FUNCTION_BLOCK ServoAxis EXTENDS ParentAxis
VAR
	
	_AxisReference				: AXIS_REF;
	
	_Enable						: MC_Power;
	_ReadStatus					: MC_ReadStatus;
	_Reset						: MC_Reset;
	_MoveRelative				: MC_MoveRelative;
	
	_Status						: NcAxisRefStatus;
	
END_VAR

METHOD CyclicUpdate : HRESULT
VAR_INPUT
END_VAR

_ClassRunningIndicatorToggle := NOT(_ClassRunningIndicatorToggle);

_Enable(Axis := _AxisReference);
_Reset(Axis := _AxisReference);
_MoveRelative(Axis := _AxisReference);

_ReadStatus
(
	Axis 					:= _AxisReference,
	Enable 					:= TRUE,
	Error 					=> _Status._Error,
	ErrorID 				=> _Status._ErrorID,
	ErrorStop 				=> _Status._ErrorStop,
	Disabled 				=> _Status._Disabled,
	Stopping 				=> _Status._Stopping,
	StandStill 				=> _Status._StandStill,
	DiscreteMotion 			=> _Status._DiscreteMotion,
	ContinuousMotion 		=> _Status._ContinuousMotion,
	SynchronizedMotion 		=> _Status._SynchronizedMotion,
	Homing 					=> _Status._Homing,
	ConstantVelocity 		=> _Status._ConstantVelocity,
	Accelerating 			=> _Status._Accelerating,
	Decelerating 			=> _Status._Decelerating,
	Status 					=> _Status._Status
);

_IsBusyMoving :=
(
	_ReadStatus.DiscreteMotion OR
	_ReadStatus.ConstantVelocity OR
	_ReadStatus.SynchronizedMotion
);

_IsBusyStopping :=
(
	_ReadStatus.Stopping
);

_IsReadyForCommand :=
(
	NOT(_ReadStatus.Disabled) AND
	NOT(_IsBusyMoving) AND
	NOT(_IsBusyStopping) AND
	NOT(_ReadStatus.Error) AND
	NOT(_ReadStatus.ErrorStop)
);

_IsDoneWithCommand :=
(
	_Reset.Done OR
	_MoveRelative.Done
);

_IsInError :=
(
	_ReadStatus.Error
);

_CurrentErrorCode := _ReadStatus.ErrorID;
	
IF _Status._ErrorID <> 0 THEN
	_PreviousErrorCode := _ReadStatus.ErrorID;
END_IF

_ErrorRTrig(CLK := _IsInError);
IF _ErrorRTrig.Q THEN
	_ErrorCount := _ErrorCount + 1;
END_IF


CyclicUpdate := 1;
RETURN;
END_METHOD

METHOD StartDisable : BOOL
_Enable(Axis := _AxisReference);

_Enable.Enable := FALSE;
_Enable.Enable_Negative := FALSE;
_Enable.Enable_Positive := FALSE;
_Enable.Override := 0;

IF NOT(_Enable.Status) THEN
	StartDisable := TRUE;
	RETURN;
ELSE
	;
END_IF

RETURN;
END_METHOD

METHOD StartEnable : BOOL
_Enable(Axis := _AxisReference);

_Enable.Enable := TRUE;
_Enable.Enable_Negative := TRUE;
_Enable.Enable_Positive := TRUE;
_Enable.Override := 100;

IF _Enable.Error THEN
	_Enable.Enable := FALSE;
	StartEnable := FALSE;
	RETURN;
ELSE
	;
END_IF

IF _Enable.Status THEN
	StartEnable := TRUE;
	RETURN;
ELSE
	;
END_IF

RETURN;
END_METHOD

METHOD StartErrorChecking : BOOL
IF _IsInError THEN
	StartErrorChecking := TRUE;
	RETURN;
ELSE
	;
END_IF

RETURN;
END_METHOD

METHOD StartMovement : BOOL
_MoveRelative(Axis := _AxisReference);
_MoveRelative.Distance := 100;
_MoveRelative.Velocity := 20;
_MoveRelative.Execute := TRUE;

IF _MoveRelative.Error THEN
	_MoveRelative.Execute := FALSE;
	StartMovement := FALSE;
	RETURN;
ELSE
	;
END_IF

IF _MoveRelative.Done THEN
	_MoveRelative.Execute := FALSE;
	StartMovement := TRUE;
	RETURN;
ELSE
	;
END_IF

RETURN;
END_METHOD

METHOD StartReset : BOOL
_MoveRelative(Axis := _AxisReference);
_Reset(Axis := _AxisReference);

_MoveRelative.Execute := FALSE;

_Reset.Execute := TRUE;

IF _Reset.Error THEN
	_Reset.Execute := FALSE;
	StartReset := FALSE;
	RETURN;
ELSE
	;
END_IF

IF _Reset.Done THEN
	_Reset.Execute := FALSE;
	StartReset := TRUE;
ELSE
	;
END_IF
END_METHOD

END_FUNCTION_BLOCK

(* stored: Version 1.1.0.1, ProductVersion 3.1.4024.12
   POU ServoAxis: Id {26452b28-7ab5-49f1-a26d-862a61902626}, SpecialFunc None
   Folder METH: Id {29812a1c-8682-40c9-b187-562c333ac7c7}
   Folder PROP: Id {95b1584f-04a4-4070-99b8-73a50df63774}
   Method CyclicUpdate: Id {cf0f58ec-dc9a-4e00-98cf-928468696fb2}
   Method StartDisable: Id {0978b676-9045-4216-aa0e-c51dea3ee422}
   Method StartEnable: Id {2b737eca-ff29-4152-bc27-b5c3e407fd90}
   Method StartErrorChecking: Id {26ea8b5e-d8b0-4411-b8b7-aecbfb9a6f13}
   Method StartMovement: Id {b63463d0-f34d-41ec-b50b-726fc4af6150}
   Method StartReset: Id {964eb855-0bd1-4c99-ad94-d1876c6d809f} *)
